GLOBALCONSTANTS SubStrings (* Global constants *)
  (* Standard: 61499-1 *)
  (* Version 1.0, 2026-08-31, Franz Höpfinger, Meisterschulen am Ostbahnhof *)
  PACKAGE Meins::InputOutputTester::Button_AI_Calibrate_OPC_UA;
  VAR_GLOBAL CONSTANT
    AIC_I1_RAW_WRITE : WSTRING := "opc_ua[WRITE;/Objects/AnalogCalibrated/I1/RAW,1:s=AIC_I1_RAW]";
    AIC_I1_CAL_WRITE : WSTRING := "opc_ua[WRITE;/Objects/AnalogCalibrated/I1/CAL,1:s=AIC_I1_CAL]";
    AIC_I2_RAW_WRITE : WSTRING := "opc_ua[WRITE;/Objects/AnalogCalibrated/I2/RAW,1:s=AIC_I2_RAW]";
    AIC_I2_CAL_WRITE : WSTRING := "opc_ua[WRITE;/Objects/AnalogCalibrated/I2/CAL,1:s=AIC_I2_CAL]";
    AIC_I3_RAW_WRITE : WSTRING := "opc_ua[WRITE;/Objects/AnalogCalibrated/I3/RAW,1:s=AIC_I3_RAW]";
    AIC_I3_CAL_WRITE : WSTRING := "opc_ua[WRITE;/Objects/AnalogCalibrated/I3/CAL,1:s=AIC_I3_CAL]";
    AIC_I4_RAW_WRITE : WSTRING := "opc_ua[WRITE;/Objects/AnalogCalibrated/I4/RAW,1:s=AIC_I4_RAW]";
    AIC_I4_CAL_WRITE : WSTRING := "opc_ua[WRITE;/Objects/AnalogCalibrated/I4/CAL,1:s=AIC_I4_CAL]";
    AIC_I5_RAW_WRITE : WSTRING := "opc_ua[WRITE;/Objects/AnalogCalibrated/I5/RAW,1:s=AIC_I5_RAW]";
    AIC_I5_CAL_WRITE : WSTRING := "opc_ua[WRITE;/Objects/AnalogCalibrated/I5/CAL,1:s=AIC_I5_CAL]";
    AIC_I6_RAW_WRITE : WSTRING := "opc_ua[WRITE;/Objects/AnalogCalibrated/I6/RAW,1:s=AIC_I6_RAW]";
    AIC_I6_CAL_WRITE : WSTRING := "opc_ua[WRITE;/Objects/AnalogCalibrated/I6/CAL,1:s=AIC_I6_CAL]";
    AIC_I7_RAW_WRITE : WSTRING := "opc_ua[WRITE;/Objects/AnalogCalibrated/I7/RAW,1:s=AIC_I7_RAW]";
    AIC_I7_CAL_WRITE : WSTRING := "opc_ua[WRITE;/Objects/AnalogCalibrated/I7/CAL,1:s=AIC_I7_CAL]";
    AIC_I8_RAW_WRITE : WSTRING := "opc_ua[WRITE;/Objects/AnalogCalibrated/I8/RAW,1:s=AIC_I8_RAW]";
    AIC_I8_CAL_WRITE : WSTRING := "opc_ua[WRITE;/Objects/AnalogCalibrated/I8/CAL,1:s=AIC_I8_CAL]";
    AIC_I1_CO_METHOD : WSTRING := "opc_ua[CREATE_METHOD;/Objects/AnalogCalibrated/I1/COMethod,1:s=AIC_I1_CO_METHOD]";
    AIC_I1_CS_METHOD : WSTRING := "opc_ua[CREATE_METHOD;/Objects/AnalogCalibrated/I1/CSMethod,1:s=AIC_I1_CS_METHOD]";
    AIC_I2_CO_METHOD : WSTRING := "opc_ua[CREATE_METHOD;/Objects/AnalogCalibrated/I2/COMethod,1:s=AIC_I2_CO_METHOD]";
    AIC_I2_CS_METHOD : WSTRING := "opc_ua[CREATE_METHOD;/Objects/AnalogCalibrated/I2/CSMethod,1:s=AIC_I2_CS_METHOD]";
    AIC_I3_CO_METHOD : WSTRING := "opc_ua[CREATE_METHOD;/Objects/AnalogCalibrated/I3/COMethod,1:s=AIC_I3_CO_METHOD]";
    AIC_I3_CS_METHOD : WSTRING := "opc_ua[CREATE_METHOD;/Objects/AnalogCalibrated/I3/CSMethod,1:s=AIC_I3_CS_METHOD]";
    AIC_I4_CO_METHOD : WSTRING := "opc_ua[CREATE_METHOD;/Objects/AnalogCalibrated/I4/COMethod,1:s=AIC_I4_CO_METHOD]";
    AIC_I4_CS_METHOD : WSTRING := "opc_ua[CREATE_METHOD;/Objects/AnalogCalibrated/I4/CSMethod,1:s=AIC_I4_CS_METHOD]";
    AIC_I5_CO_METHOD : WSTRING := "opc_ua[CREATE_METHOD;/Objects/AnalogCalibrated/I5/COMethod,1:s=AIC_I5_CO_METHOD]";
    AIC_I5_CS_METHOD : WSTRING := "opc_ua[CREATE_METHOD;/Objects/AnalogCalibrated/I5/CSMethod,1:s=AIC_I5_CS_METHOD]";
    AIC_I6_CO_METHOD : WSTRING := "opc_ua[CREATE_METHOD;/Objects/AnalogCalibrated/I6/COMethod,1:s=AIC_I6_CO_METHOD]";
    AIC_I6_CS_METHOD : WSTRING := "opc_ua[CREATE_METHOD;/Objects/AnalogCalibrated/I6/CSMethod,1:s=AIC_I6_CS_METHOD]";
    AIC_I7_CO_METHOD : WSTRING := "opc_ua[CREATE_METHOD;/Objects/AnalogCalibrated/I7/COMethod,1:s=AIC_I7_CO_METHOD]";
    AIC_I7_CS_METHOD : WSTRING := "opc_ua[CREATE_METHOD;/Objects/AnalogCalibrated/I7/CSMethod,1:s=AIC_I7_CS_METHOD]";
    AIC_I8_CO_METHOD : WSTRING := "opc_ua[CREATE_METHOD;/Objects/AnalogCalibrated/I8/COMethod,1:s=AIC_I8_CO_METHOD]";
    AIC_I8_CS_METHOD : WSTRING := "opc_ua[CREATE_METHOD;/Objects/AnalogCalibrated/I8/CSMethod,1:s=AIC_I8_CS_METHOD]";
    Q01_READ : WSTRING := "opc_ua[READ;/Objects/DigitalOutput/Q01,1:s=Q01]";
    Q01_WRITE : WSTRING := "opc_ua[WRITE;/Objects/DigitalOutput/Q01,1:s=Q01]";
    Q02_READ : WSTRING := "opc_ua[READ;/Objects/DigitalOutput/Q02,1:s=Q02]";
    Q02_WRITE : WSTRING := "opc_ua[WRITE;/Objects/DigitalOutput/Q02,1:s=Q02]";
    Q03_READ : WSTRING := "opc_ua[READ;/Objects/DigitalOutput/Q03,1:s=Q03]";
    Q03_WRITE : WSTRING := "opc_ua[WRITE;/Objects/DigitalOutput/Q03,1:s=Q03]";
    Q04_READ : WSTRING := "opc_ua[READ;/Objects/DigitalOutput/Q04,1:s=Q04]";
    Q04_WRITE : WSTRING := "opc_ua[WRITE;/Objects/DigitalOutput/Q04,1:s=Q04]";
    Q05_READ : WSTRING := "opc_ua[READ;/Objects/DigitalOutput/Q05,1:s=Q05]";
    Q05_WRITE : WSTRING := "opc_ua[WRITE;/Objects/DigitalOutput/Q05,1:s=Q05]";
    Q06_READ : WSTRING := "opc_ua[READ;/Objects/DigitalOutput/Q06,1:s=Q06]";
    Q06_WRITE : WSTRING := "opc_ua[WRITE;/Objects/DigitalOutput/Q06,1:s=Q06]";
    Q07_READ : WSTRING := "opc_ua[READ;/Objects/DigitalOutput/Q07,1:s=Q07]";
    Q07_WRITE : WSTRING := "opc_ua[WRITE;/Objects/DigitalOutput/Q07,1:s=Q07]";
    Q08_READ : WSTRING := "opc_ua[READ;/Objects/DigitalOutput/Q08,1:s=Q08]";
    Q08_WRITE : WSTRING := "opc_ua[WRITE;/Objects/DigitalOutput/Q08,1:s=Q08]";
    Q09_READ : WSTRING := "opc_ua[READ;/Objects/DigitalOutput/Q09,1:s=Q09]";
    Q09_WRITE : WSTRING := "opc_ua[WRITE;/Objects/DigitalOutput/Q09,1:s=Q09]";
    Q10_READ : WSTRING := "opc_ua[READ;/Objects/DigitalOutput/Q10,1:s=Q10]";
    Q10_WRITE : WSTRING := "opc_ua[WRITE;/Objects/DigitalOutput/Q10,1:s=Q10]";
    Q11_READ : WSTRING := "opc_ua[READ;/Objects/DigitalOutput/Q11,1:s=Q11]";
    Q11_WRITE : WSTRING := "opc_ua[WRITE;/Objects/DigitalOutput/Q11,1:s=Q11]";
    Q12_READ : WSTRING := "opc_ua[READ;/Objects/DigitalOutput/Q12,1:s=Q12]";
    Q12_WRITE : WSTRING := "opc_ua[WRITE;/Objects/DigitalOutput/Q12,1:s=Q12]";
    Tick_WRITE : WSTRING := "opc_ua[WRITE;/Objects/System/Tick,1:s=System.Tick]";
    AIC_I1_ZERO_READ : WSTRING := "opc_ua[READ;/Objects/AnalogCalibrated/I1/ZEROExt,1:s=AIC_I1_ZERO_EXT]";
    AIC_I1_ZERO_WRITE : WSTRING := "opc_ua[WRITE;/Objects/AnalogCalibrated/I1/ZERO,1:s=AIC_I1_ZERO]";
    AIC_I1_SPAN_READ : WSTRING := "opc_ua[READ;/Objects/AnalogCalibrated/I1/SPANExt,1:s=AIC_I1_SPAN_EXT]";
    AIC_I1_SPAN_WRITE : WSTRING := "opc_ua[WRITE;/Objects/AnalogCalibrated/I1/SPAN,1:s=AIC_I1_SPAN]";
    AIC_I2_ZERO_READ : WSTRING := "opc_ua[READ;/Objects/AnalogCalibrated/I2/ZEROExt,1:s=AIC_I2_ZERO_EXT]";
    AIC_I2_ZERO_WRITE : WSTRING := "opc_ua[WRITE;/Objects/AnalogCalibrated/I2/ZERO,1:s=AIC_I2_ZERO]";
    AIC_I2_SPAN_READ : WSTRING := "opc_ua[READ;/Objects/AnalogCalibrated/I2/SPANExt,1:s=AIC_I2_SPAN_EXT]";
    AIC_I2_SPAN_WRITE : WSTRING := "opc_ua[WRITE;/Objects/AnalogCalibrated/I2/SPAN,1:s=AIC_I2_SPAN]";
    AIC_I3_ZERO_READ : WSTRING := "opc_ua[READ;/Objects/AnalogCalibrated/I3/ZEROExt,1:s=AIC_I3_ZERO_EXT]";
    AIC_I3_ZERO_WRITE : WSTRING := "opc_ua[WRITE;/Objects/AnalogCalibrated/I3/ZERO,1:s=AIC_I3_ZERO]";
    AIC_I3_SPAN_READ : WSTRING := "opc_ua[READ;/Objects/AnalogCalibrated/I3/SPANExt,1:s=AIC_I3_SPAN_EXT]";
    AIC_I3_SPAN_WRITE : WSTRING := "opc_ua[WRITE;/Objects/AnalogCalibrated/I3/SPAN,1:s=AIC_I3_SPAN]";
    AIC_I4_ZERO_READ : WSTRING := "opc_ua[READ;/Objects/AnalogCalibrated/I4/ZEROExt,1:s=AIC_I4_ZERO_EXT]";
    AIC_I4_ZERO_WRITE : WSTRING := "opc_ua[WRITE;/Objects/AnalogCalibrated/I4/ZERO,1:s=AIC_I4_ZERO]";
    AIC_I4_SPAN_READ : WSTRING := "opc_ua[READ;/Objects/AnalogCalibrated/I4/SPANExt,1:s=AIC_I4_SPAN_EXT]";
    AIC_I4_SPAN_WRITE : WSTRING := "opc_ua[WRITE;/Objects/AnalogCalibrated/I4/SPAN,1:s=AIC_I4_SPAN]";
    AIC_I5_ZERO_READ : WSTRING := "opc_ua[READ;/Objects/AnalogCalibrated/I5/ZEROExt,1:s=AIC_I5_ZERO_EXT]";
    AIC_I5_ZERO_WRITE : WSTRING := "opc_ua[WRITE;/Objects/AnalogCalibrated/I5/ZERO,1:s=AIC_I5_ZERO]";
    AIC_I5_SPAN_READ : WSTRING := "opc_ua[READ;/Objects/AnalogCalibrated/I5/SPANExt,1:s=AIC_I5_SPAN_EXT]";
    AIC_I5_SPAN_WRITE : WSTRING := "opc_ua[WRITE;/Objects/AnalogCalibrated/I5/SPAN,1:s=AIC_I5_SPAN]";
    AIC_I6_ZERO_READ : WSTRING := "opc_ua[READ;/Objects/AnalogCalibrated/I6/ZEROExt,1:s=AIC_I6_ZERO_EXT]";
    AIC_I6_ZERO_WRITE : WSTRING := "opc_ua[WRITE;/Objects/AnalogCalibrated/I6/ZERO,1:s=AIC_I6_ZERO]";
    AIC_I6_SPAN_READ : WSTRING := "opc_ua[READ;/Objects/AnalogCalibrated/I6/SPANExt,1:s=AIC_I6_SPAN_EXT]";
    AIC_I6_SPAN_WRITE : WSTRING := "opc_ua[WRITE;/Objects/AnalogCalibrated/I6/SPAN,1:s=AIC_I6_SPAN]";
    AIC_I7_ZERO_READ : WSTRING := "opc_ua[READ;/Objects/AnalogCalibrated/I7/ZEROExt,1:s=AIC_I7_ZERO_EXT]";
    AIC_I7_ZERO_WRITE : WSTRING := "opc_ua[WRITE;/Objects/AnalogCalibrated/I7/ZERO,1:s=AIC_I7_ZERO]";
    AIC_I7_SPAN_READ : WSTRING := "opc_ua[READ;/Objects/AnalogCalibrated/I7/SPANExt,1:s=AIC_I7_SPAN_EXT]";
    AIC_I7_SPAN_WRITE : WSTRING := "opc_ua[WRITE;/Objects/AnalogCalibrated/I7/SPAN,1:s=AIC_I7_SPAN]";
    AIC_I8_ZERO_READ : WSTRING := "opc_ua[READ;/Objects/AnalogCalibrated/I8/ZEROExt,1:s=AIC_I8_ZERO_EXT]";
    AIC_I8_ZERO_WRITE : WSTRING := "opc_ua[WRITE;/Objects/AnalogCalibrated/I8/ZERO,1:s=AIC_I8_ZERO]";
    AIC_I8_SPAN_READ : WSTRING := "opc_ua[READ;/Objects/AnalogCalibrated/I8/SPANExt,1:s=AIC_I8_SPAN_EXT]";
    AIC_I8_SPAN_WRITE : WSTRING := "opc_ua[WRITE;/Objects/AnalogCalibrated/I8/SPAN,1:s=AIC_I8_SPAN]";
  END_VAR
END_GLOBALCONSTANTS
